FUNCTION_BLOCK OneStateTest
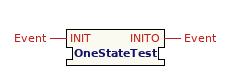
  EVENT_INPUT
    INIT;
  END_EVENT
  EVENT_OUTPUT
    INITO;
  END_EVENT
  EC_STATES
    START;
  END_STATES
  ALGORITHM NewAlgorithm1 IN ST:

  END_ALGORITHM
  ALGORITHM  IN ST:

  END_ALGORITHM
END_FUNCTION_BLOCK
